SYSTEM NestedStructRenameTest
  (* Version 1.0, 2026-07-21, Dimitrios Kalligaridis *)
  APPLICATION App
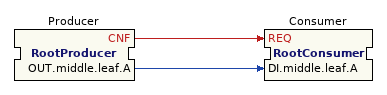
    FBS
      Producer : RootProducer(OUT.middle.leaf.A :=  {SET_ATTRIBUTE(TestAttribute, 42)});
      Consumer : RootConsumer;
    END_FBS
    EVENT_CONNECTIONS
      Producer.CNF TO Consumer.REQ;
    END_CONNECTIONS
    DATA_CONNECTIONS
      Producer.OUT.middle.leaf.A TO Consumer.DI.middle.leaf.A;
    END_CONNECTIONS
  END_APPLICATION
END_SYSTEM
